{attribute 'qualified_only'}
VAR_GLOBAL

    // ==================================================
    // DIGITALE EINGÄNGE
    // ==================================================

    DI_NotHaltFrei        AT %I* : BOOL;
    DI_SchutzhaubeZu      AT %I* : BOOL;
    DI_PaletteEingang     AT %I* : BOOL;
    DI_PalettePositioniert AT %I* : BOOL;
    DI_HubUnten           AT %I* : BOOL;
    DI_HubOben            AT %I* : BOOL;
    DI_KollisionFrei      AT %I* : BOOL;
    DI_WerkerQuittierung  AT %I* : BOOL;


    // ==================================================
    // DIGITALE AUSGÄNGE
    // ==================================================

    DO_SignalGruen        AT %Q* : BOOL;
    DO_AlarmRot           AT %Q* : BOOL;
    DO_Foerderband        AT %Q* : BOOL;
    DO_FoerderbandStopp   AT %Q* : BOOL;
    DO_HubwerkHoch        AT %Q* : BOOL;
    DO_HubwerkRunter      AT %Q* : BOOL;
    DO_ProzessFreigabe    AT %Q* : BOOL;
    DO_Heizfreigabe       AT %Q* : BOOL;


    // ==================================================
    // ANALOGE EINGÄNGE
    // ==================================================

    AI_FolienTemperatur   AT %I* : REAL;
    AI_MotorTemperatur    AT %I* : REAL;

	// ==================================================
	// INTERNE PROGRAMMVARIABLEN
	// ==================================================
	
	Schritt : INT := 0;
	AlarmAktiv : BOOL := FALSE;


END_VAR

(* stored: Version 1.1.0.1, ProductVersion 3.1.4024.16
   GVL GVL_IO: Id {bed1bbdf-fede-4f6f-921a-dd02debe56d0} *)
